{attribute 'GeneratedUsingTerminal: EJ1918-0000-0017'}
{attribute addProperty BoxType "EJ1918-0000-0017"}
{attribute addProperty Id "EtcSlaveTerminalBaseModule_1_FSOEModule_1_FSOE_18ED951F26Module_2_DEVICEIOModule_2_DEVICEIO_5FA6B4E72Module_3_FSLOGICModule_3_FSLOGIC_DEAB45222WcStateAT %I*WcState_9091E0EB2InfoDataAT %I*InfoData_32EB74EA10"}
{attribute addProperty CRC "3089978320"}
{attribute addProperty Size "42"}
TYPE EJ1918_B82D53D0 EXTENDS EtcSlaveTerminalBase :
STRUCT
	{attribute addProperty Name "Module_1_FSOE"}
	Module_1_FSOE : Module_1_FSOE_18ED951F;
	{attribute addProperty Name "Module_2_DEVICEIO"}
	Module_2_DEVICEIO : Module_2_DEVICEIO_5FA6B4E7;
	{attribute addProperty Name "Module_3_FSLOGIC"}
	Module_3_FSLOGIC : Module_3_FSLOGIC_DEAB4522;
	{attribute addProperty Name "WcState"}
	WcState : WcState_9091E0EB;
	{attribute addProperty Name "InfoData"}
	InfoData : InfoData_32EB74EA;
END_STRUCT
END_TYPE

(* stored: Version 1.2.0.0, ProductVersion 3.1.4024.9
   DUT EJ1918_B82D53D0: Id {aa3a823d-bf1b-4a56-85a2-ba2f15f1661d} *)
